(* CoDeSys 2.3.9.35 project: poka-yoke.pro *)
(* Author: Altus *)
(* Libraries: DU35x.lib 7.7.11 15:59:13, Navigation.lib 15.7.11 10:06:00, SysLibTargetVisu.lib 26.11.08 09:53:28, Standard.lib 26.11.08 09:46:20, Iecsfc.lib 26.11.08 09:46:14, SYSLIBCALLBACK.LIB 26.11.08 09:53:30 *)

(* PLC configuration (modules and I/O channels)
COM1 [COM1] node 0, in %IB0 out %QB0 {BaudRate = 115200; Paridade = Sem Paridade; StopBits = 1 Stop Bit; Modem = Sem RTS/CTS; Delay = 5}
  MToolIEC [Codesys] node 0, in %IB0 out %QB0
COM2 [COM2] node 1, in %IB0 out %QB0 {BaudRate = 115200; Paridade = Sem Paridade; StopBits = 1 Stop Bit; Modem = Sem RTS/CTS; Delay = 5}
  Desabilitada [Desabilitado485] node 0, in %IB0 out %QB0
Entradas Digitais 0 [Entradas0] node 0, in %IW0 out %QB0
  I00 AT %IX0.0 [BitInput] I0.0
  I01 AT %IX0.1 [BitInput] I0.1
  I02 AT %IX0.2 [BitInput] I0.2
  I03 AT %IX0.3 [BitInput] I0.3
  I04 AT %IX0.4 [BitInput] I0.4
  I05 AT %IX0.5 [BitInput] I0.5
  I06 AT %IX0.6 [BitInput] I0.6
  I07 AT %IX0.7 [BitInput] I0.7
  I08 AT %IX0.8 [BitInput] I0.8
Entradas Digitais 1 [Entradas1] node 0, in %IW1 out %QB0
  I10 AT %IX1.0 [BitInput] I1.0
  I11 AT %IX1.1 [BitInput] I1.1
  I12 AT %IX1.2 [BitInput] I1.2
  I13 AT %IX1.3 [BitInput] I1.3
  I14 AT %IX1.4 [BitInput] I1.4
  I15 AT %IX1.5 [BitInput] I1.5
  I16 AT %IX1.6 [BitInput] I1.6
  I17 AT %IX1.7 [BitInput] I1.7
  I18 AT %IX1.8 [BitInput] I1.8
I20 AT %IX2.0 [BitInput] I2.0
I21 AT %IX2.1 [BitInput] I2.1
AI0 AT %IW4 [WordInput] AI0 {TipoAnalogica = Channel Disable; FiltroAnalogica = Filter 0 - AI=2ms  / AV=90ms; FundoEscala = 0}
AI1 AT %IW5 [WordInput] AI1 {TipoAnalogica = Channel Disable; FiltroAnalogica = Filter 0 - AI=2ms  / AV=90ms; FundoEscala = 0}
AI2 AT %IW6 [WordInput] AI2 {TipoAnalogica = Channel Disable; FiltroAnalogica = Filter 0 - AI=2ms  / AV=90ms; FundoEscala = 0}
AI3 AT %IW7 [WordInput] AI3 {TipoAnalogica = Channel Disable; FiltroAnalogica = Filter 0 - AI=2ms  / AV=90ms; FundoEscala = 0}
Entradas Rápidas [EntradasRapidas] node 1, in %IB16 out %QB0
  Bloco 0 [Bloco0] node 0, in %IB16 out %QB0
    Desabilitado [DesabilitadoBloco0] node 0, in %IB16 out %QB0
  Bloco 1 [Bloco1] node 1, in %IB16 out %QB0
    Desabilitado [DesabilitadoBloco1] node 0, in %IB16 out %QB0
  Entrada Configuravél Bloco 0 [EntradaConfiBloco0] node 2, in %IB16 out %QB0
    Contador 0 [EntradaConfContador0] node 0, in %IB16 out %QB0 {EntradaConfiguravelContador = Disable}
  Entrada Configuravél Bloco 1 [EntradaConfiBloco1] node 3, in %IB16 out %QB0
    Contador 2 [EntradaConfContador2] node 0, in %IB16 out %QB0 {EntradaConfiguravelContador = Disable}
Saídas [Saidas] node 1, in %IB13 out %QB0
  Saídas Digitais 0 [Saidas0] node 0, in %IW0 out %QW0
    Q00 AT %QX0.0 [BitOutput] Q0.0
    Q01 AT %QX0.1 [BitOutput] Q0.1
    Q02 AT %QX0.2 [BitOutput] Q0.2
    Q03 AT %QX0.3 [BitOutput] Q0.3
    Q04 AT %QX0.4 [BitOutput] Q0.4
    Q05 AT %QX0.5 [BitOutput] Q0.5
    Q06 AT %QX0.6 [BitOutput] Q0.6
    Q07 AT %QX0.7 [BitOutput] Q0.7
  Saídas Digitais 1 [Saidas1] node 0, in %IW0 out %QW1
    Q10 AT %QX1.0 [BitOutput] Q1.0
    Q11 AT %QX1.1 [BitOutput] Q1.1
    Q12 AT %QX1.2 [BitOutput] Q1.2
    Q13 AT %QX1.3 [BitOutput] Q1.3
    Q14 AT %QX1.4 [BitOutput] Q1.4
    Q15 AT %QX1.5 [BitOutput] Q1.5
    Q16 AT %QX1.6 [BitOutput] Q1.6
    Q17 AT %QX1.7 [BitOutput] Q1.7
  Saídas Analógicas [SaidaAnalogica] node 0, in %IW0 out %QW3
    AO0 AT %QW3 [WordOutput] AO0 {TipoAnalogica = Channel Disable; FundoEscala = 0}
    AO1 AT %QW4 [WordOutput] AO1 {TipoAnalogica = Channel Disable; FundoEscala = 0}
  Saídas Rápidas [SaidasRapidas] node 1, in %IB0 out %QB10
    Saída Rápida 0 Desabilitada [DesabilitadoF0] node 0, in %IB0 out %QB10
    Saída Rápida 1 Desabilitada [DesabilitadoF1] node 1, in %IB0 out %QB10
  Saídas Comum de Contador [SaidasContador] node 2, in %IB0 out %QB10
    Saída do Bloco 0 Desabilitada [DesabilitadoSaidaBloco0] node 0, in %IB0 out %QB10
    Saída do Bloco 1 Desabilitada [DesabilitadoSaidaBloco1] node 1, in %IB0 out %QB10
Eventos Externos [Eventos] node 2, in %IB13 out %QB6
  Evento Temporizado [TimerEvent] node 0, in %IB13 out %QB6 {Intervalo = 10}
*)

(* Task configuration *)
TASK PRINCIPAL (PRIORITY := 1, INTERVAL := T#1ms);
	PLC_PRG();
END_TASK
TASK NAVIGATION (PRIORITY := 1, INTERVAL := T#20ms);
	NAVEGA();
END_TASK
TASK VISUALIZATION (PRIORITY := 1, INTERVAL := T#500ms);
	MAINTARGETVISU_PAINT_CODE
END_TASK
TASK KEYBOARD_USAGE (PRIORITY := 1, INTERVAL := T#20ms);
	MAINTARGETVISU_INPUT_CODE
END_TASK

(* Global variable list: Variáveis globais *)
(*CONSTANTES*)
VAR_GLOBAL CONSTANT
	NUMMAX_SENSORES: USINT := 14; (* NUMERO MAXIMO DE SENSORES *)
	NUMMAX_PARAFUSA: USINT := 1;
	NUMMAX_PROGBITS: USINT := 4;
	NUMMAX_MODELOS: USINT := 15;
	NUMMAX_SAIDAS: USINT := 14;
	NUM_ETAPAS: USINT := 12;
	NUM_ATIVOS: USINT := 4;
	SEGURANCA_ENABLED: BOOL := TRUE;
	CODE_PARAFUSA: USINT := 15;
	CODE_KEY_F: ARRAY [1..7] OF USINT := 16#70, 16#71, 16#72, 16#73, 16#74, 16#75, 16#76;
	CODE_KEY_MAIN: USINT := 16#24;
	CODE_KEY_UP: USINT := 16#26;
	CODE_KEY_DOWN: USINT := 16#28;
	CODE_KEY_DOT: USINT := 16#2E;
	CODE_KEY_ZERO: USINT := 16#30;
	CODE_KEY_ESC: USINT := 16#1B;
END_VAR

(*VARS GERAIS*)
VAR_GLOBAL
	PRIMEIRO_STEP: BOOL := TRUE;
	SEGUNDO_STEP: BOOL;
	TERCEIRO_STEP: BOOL;
	QUARTO_STEP: BOOL;
	QUINTO_STEP: BOOL;
	SEXTO_STEP: BOOL;
	SETIMO_STEP: BOOL;
	OITAVO_STEP: BOOL;
	NONO_STEP: BOOL;
	DECIMO_STEP: BOOL;
	ONZE_STEP: BOOL;
	DOZE_STEP: BOOL;
	TREZE_STEP: BOOL;
	QUATORZE_STEP: BOOL;
	QUINZE_STEP: BOOL;
	MODELOS_CONFIG4: BOOL;
	MODELOS_RANGE: USINT := 0;
	X: USINT := 1;
	Y: USINT := 1;
	Z: USINT := 1;
	IHM_X: USINT := 1;
	IHM_STRING_TITLE: STRING(20);
	IHM_STRING_DESCRIPTION: STRING(30);
	IHM_NUMMAX_SENSORES: USINT;
	IHM_NUMMAX_PARAFUSA: USINT;
	IHM_NUMMAX_PROGBITS: USINT;
	IHM_NUMMAX_PROGS: USINT;
	IHM_BLOQUEIA_PROGBITS: BOOL;
	IHM_BLOQUEIA_MODELOS: ARRAY [1..4] OF BOOL;
	IHM_ESCONDER_ZERAR: BOOL;
	IHM_ESCONDER_RESET: BOOL;
	IHM_ESCONDER_SETUP: BOOL;
	IHM_ESCONDER_MODELOS: ARRAY [1..4] OF BOOL;
	IHM_ESCONDER_MODELO4BACK: BOOL;
	IHM_ENTRADA_PROGS: BOOL;
	IHM_INT_ETAPAS: USINT;
	IHM_INT_ATIVOS: ARRAY [1..4] OF USINT;
	TECLA_F: ARRAY [1..7] OF BOOL;
	TECLA_MAIN: BOOL;
	TECLA_UP: BOOL;
	TECLA_DOWN: BOOL;
	TECLA_DOT: BOOL;
	TECLA_ZERO: BOOL;
	TECLA_ESC: BOOL;
	PASS_LIBERADO: BOOL;
	IHM_STRING_CHAVE: STRING(3);
	IHM_INT_SENHA: USINT;
	SENHA_GERADA : USINT;
	IHM_STRING_MODELOS: ARRAY [1..4] OF INT;
	MODELO_SELECIONADO: INT;

	(*MIGRADOS*)
	PRONTO: USINT;
	ARRAY_SENSORES_IN: ARRAY [1..NUMMAX_SENSORES] OF BOOL;
	ARRAY_SENSORES_OUT: ARRAY [1..NUMMAX_SENSORES] OF BOOL;
	ARRAY_SENSORES_OLDSTATE: ARRAY [1..NUMMAX_SENSORES] OF BOOL;
	ARRAY_DE_ATIVOS: ARRAY [1..NUM_ATIVOS] OF USINT;
	ARRAY_PROGBYTE_PARAFUSA: ARRAY [1..4] OF BOOL;
END_VAR

(*RETENTIVAS*)
VAR_GLOBAL RETAIN
	PRIMEIRO_START: BOOL := TRUE;
	NUM_SENSORES: USINT;
	NUM_PARAFUSA: USINT;
	NUM_PROGBITS: USINT;
	NUM_MODELOS: USINT;
	MATRIZ: ARRAY [1..NUMMAX_MODELOS, 1..NUM_ETAPAS, 1..NUM_ATIVOS] OF USINT;
	MODELOS: ARRAY [1..NUMMAX_MODELOS] OF INT;
END_VAR

(*VARS DE ENTRADA*)
VAR_GLOBAL (*--------VARIAVEIS DE ENTRADA-------*)
	KAP_IN 		AT %IX0.0: BOOL;
	SENSOR1_IN 	AT %IX0.1: BOOL;
	SENSOR2_IN 	AT %IX0.2: BOOL;
	SENSOR3_IN 	AT %IX0.3: BOOL;
	SENSOR4_IN 	AT %IX0.4: BOOL;
	SENSOR5_IN 	AT %IX0.5: BOOL;
	SENSOR6_IN 	AT %IX0.6: BOOL;
	SENSOR7_IN 	AT %IX0.7: BOOL;
	SENSOR8_IN 	AT %IX1.0: BOOL;
	SENSOR9_IN 	AT %IX1.1: BOOL;
	SENSOR10_IN AT %IX1.2: BOOL;
	TORQUEOK_IN AT %IX2.0: BOOL;
	TORQUENOK_IN AT %IX2.1: BOOL;
END_VAR

(*VARS DE SAIDA*)
VAR_GLOBAL
	SENSOR1_OUT AT %QX0.1: BOOL;
	SENSOR2_OUT AT %QX0.2: BOOL;
	SENSOR3_OUT AT %QX0.3: BOOL;
	SENSOR4_OUT AT %QX0.4: BOOL;
	SENSOR5_OUT AT %QX0.5: BOOL;
	SENSOR6_OUT AT %QX0.6: BOOL;
	SENSOR7_OUT AT %QX0.7: BOOL;
	SENSOR8_OUT AT %QX1.0: BOOL;
	SENSOR9_OUT AT %QX1.1: BOOL;
	SENSOR10_OUT AT %QX1.2: BOOL;
	PARAFUSA_ENABLE_OUT AT %QX1.3: BOOL;
	PARAFUSA_PROG1_OUT AT %QX1.4: BOOL;
	PARAFUSA_PROG2_OUT AT %QX1.5: BOOL;
	PARAFUSA_PROG3_OUT AT %QX1.6: BOOL;
	PARAFUSA_RESET_OUT AT %QX1.7: BOOL;
END_VAR

(* POU PLC_PRG, ST *)
PROGRAM PLC_PRG
VAR
	J: USINT; (* VAR USADA PARA LOOPS *)
	K: USINT; (* VAR USADA PARA LOOPS *)
	COUNT: USINT; (* VAR USADA PARA CONTAGENS *)
	NUMERO_ALEATORIO: USINT := 1;
	LETRA_ALEATORIA: STRING(1);
	NUMERO_2 : USINT := 10;
END_VAR

(*--INSTRUCOES DE MODIFICACAO
	EXPLICACOES DA PROGRAMACAO 
	COMENTARIOS ------------->*)
(*PRIMEIRA INICIALIZACAO - alternado*)
IF PRIMEIRO_STEP = TRUE  THEN
	IF PRIMEIRO_START = TRUE THEN
		IF J < 2 THEN (*RODA DUAS VEZES A INICIALIZACAO PARA GARANTIR*)
			PRG_INICIALIZA_VARS();
			CHANGE_SCREEN(ENABLE:=TRUE, VISU_NAME:='FIRST');
			J:= J +1;
		END_IF
		IF FUN_SCREEN_FIRST() = TRUE THEN
			PRIMEIRO_START := FALSE;
			CHANGE_SCREEN(ENABLE:=TRUE, VISU_NAME:='MAIN');
		END_IF
	ELSE
		PRIMEIRO_STEP := FALSE;
		SEGUNDO_STEP := TRUE;
		OITAVO_STEP := TRUE; (*talvez*)
		TECLA_F[4] := TRUE;
	END_IF
END_IF

(*CONFIGURA TELA MAIN - alternado*)
IF SEGUNDO_STEP = TRUE THEN
	(*ESCONDE BOTOES DE CONTROLE
	IHM_ESCONDER_ZERAR:= TRUE;
	IHM_ESCONDER_RESET:= TRUE;*)
	(*DEFINE OS MODELOS NA IHM*)
	FOR J:=1 TO 4 BY 1 DO
		IF J+MODELOS_RANGE <= NUM_MODELOS THEN
			IHM_STRING_MODELOS[J]:=MODELOS[J+MODELOS_RANGE];
		ELSE
			IHM_STRING_MODELOS[J]:=0;
		END_IF
	END_FOR
	(*ESCONDE OU MOSTRA O MODELO[4] NA IHM*)
	IF NUM_MODELOS = 4 THEN
		IHM_ESCONDER_MODELOS[4]:=FALSE;
		IHM_ESCONDER_MODELO4BACK:=FALSE;
		MODELOS_CONFIG4:=TRUE;
	ELSIF NUM_MODELOS > 4 THEN
		IHM_ESCONDER_MODELOS[4]:=TRUE;
		IHM_ESCONDER_MODELO4BACK:=TRUE;
		MODELOS_CONFIG4:=FALSE;
	ELSE
		IHM_ESCONDER_MODELOS[4]:=FALSE;
		IHM_ESCONDER_MODELO4BACK:=FALSE;
		MODELOS_CONFIG4:=FALSE;
	END_IF
	(*BLOQUEIA ENTRADA MODELOS IHM*)
	FOR J:=1 TO 4 BY 1 DO
		IHM_BLOQUEIA_MODELOS[J] := TRUE;
	END_FOR
	(*AVANÇA*)
	SEGUNDO_STEP:=FALSE;
	TERCEIRO_STEP:=TRUE;
	CHANGE_SCREEN(ENABLE:=TRUE, VISU_NAME:='PASS'); (*PARA DESBUGAR*)
	CHANGE_SCREEN(ENABLE:=TRUE, VISU_NAME:='MAIN'); (*ERRO DO CLP*)
	(*temp*)
	OITAVO_STEP := TRUE;
END_IF

(*VERIFICA KAP - continuo*)
IF TERCEIRO_STEP = TRUE THEN
	IF KAP_IN = TRUE THEN	(*= FALSE*)
		(*pausa tudo*)
		QUINZE_STEP := TRUE;
		IHM_STRING_TITLE := 'CONECTE';
		IHM_STRING_DESCRIPTION := 'KAP';
		IHM_ESCONDER_ZERAR:=TRUE;
		IHM_ESCONDER_RESET:=TRUE;
		IHM_ESCONDER_SETUP:=TRUE;
		QUINTO_STEP:=FALSE;
		SEXTO_STEP:=FALSE;
		NONO_STEP :=FALSE;
		DECIMO_STEP := FALSE;
	ELSE
		QUINTO_STEP := TRUE;
		SEXTO_STEP:=TRUE;
	END_IF
END_IF

(*ESCOLHA DO MODELO - continuo*)
IF QUINTO_STEP = TRUE THEN
	(*MOSTRA MAIS MODELOS*)
	IF IHM_ESCONDER_MODELO4BACK = TRUE THEN
		IF IsKeyPressed(CODE_KEY_F[7],0,0) = TRUE OR TECLA_F[7] = TRUE(*temp*) THEN
			IF MODELOS_RANGE < NUM_MODELOS -3 THEN
				MODELOS_RANGE := MODELOS_RANGE + 3;
			ELSE
				MODELOS_RANGE := 0;
			END_IF
			SEGUNDO_STEP:=TRUE;
		END_IF
	END_IF
	(*SELECIONA O MODELO*)
	FOR J:=1 TO 4 BY 1 DO
		IF IsKeyPressed(CODE_KEY_F[J+3],0,0) = TRUE OR TECLA_F[J+3] = TRUE(*temp*) THEN
			IF IHM_ESCONDER_MODELOS[J] = FALSE AND IHM_STRING_MODELOS[J] <> 0 THEN
				MODELO_SELECIONADO := IHM_STRING_MODELOS[J];
				IHM_ESCONDER_MODELOS[IHM_X] := FALSE;
				IHM_ESCONDER_MODELOS[J] := TRUE;
				IHM_X := J;
				X:= IHM_X + MODELOS_RANGE;
				Y:= 1;
				OITAVO_STEP := TRUE;
				PRG_SENSORES.DESATIVAR_TODOS();
				PRG_PARAFUSA.DESATIVAR();
				EXIT;
			END_IF
		END_IF
	END_FOR

	(*DESTACA MODELO SELECIONADO NA IHM*)
	IF MODELO_SELECIONADO <> IHM_STRING_MODELOS[IHM_X] THEN
		IHM_ESCONDER_MODELOS[IHM_X] := FALSE;
	ELSE
		IHM_ESCONDER_MODELOS[IHM_X] := TRUE;
	END_IF
	(*RESETA TECLAS - temp*)
	FOR J:=4 TO 7 BY 1 DO
		TECLA_F[J] := FALSE;(*temp*)
	END_FOR
END_IF

(*VERIFICA TECLAS DE CONTROLE - continuo*)
IF SEXTO_STEP = TRUE THEN
	IF IsKeyPressed(CODE_KEY_F[1],0,0) = TRUE OR TECLA_F[1] = TRUE(*temp*) THEN
		IF IHM_ESCONDER_ZERAR = FALSE THEN
			(*zera o ciclo*)
			PRG_SENSORES.DESATIVAR_TODOS();
			PRG_PARAFUSA.DESATIVAR();
			Y:= 1;
			OITAVO_STEP := TRUE;
		END_IF
		TECLA_F[1] := FALSE;(*temp*)
	END_IF
	IF IsKeyPressed(CODE_KEY_F[2],0,0) = TRUE OR TECLA_F[2] = TRUE(*temp*) THEN
		IF IHM_ESCONDER_RESET = FALSE THEN
			(*reseta do pause na etapa*)
			TERCEIRO_STEP := TRUE;
			QUINTO_STEP := TRUE;
			SEXTO_STEP := TRUE;
			DECIMO_STEP := TRUE;
		END_IF
		TECLA_F[2] := FALSE;(*temp*)
	END_IF
	IF IsKeyPressed(CODE_KEY_F[3],0,0) = TRUE OR TECLA_F[3] = TRUE(*temp*) THEN
		IF IHM_ESCONDER_SETUP = FALSE THEN
			(*desliga tudo e zera*)
			TERCEIRO_STEP := FALSE;
			QUINTO_STEP := FALSE;
			SEXTO_STEP := FALSE;
			(*vai para a tela PASS*)
			IF NUMERO_2 = 10 THEN
				LETRA_ALEATORIA := 'A';
			ELSIF NUMERO_2 = 11 THEN
				LETRA_ALEATORIA := 'B';
			ELSIF NUMERO_2 = 12 THEN
				LETRA_ALEATORIA := 'C';
			ELSIF NUMERO_2 = 13 THEN
				LETRA_ALEATORIA := 'D';
			ELSIF NUMERO_2 = 14 THEN
				LETRA_ALEATORIA := 'E';
			ELSIF NUMERO_2 = 15 THEN
				LETRA_ALEATORIA := 'F';
			END_IF
			IHM_STRING_CHAVE:= CONCAT(USINT_TO_STRING(NUMERO_ALEATORIO),LETRA_ALEATORIA);
			IHM_INT_SENHA := 0;
			SENHA_GERADA := NUMERO_ALEATORIO * NUMERO_2;
			CHANGE_SCREEN(ENABLE:=TRUE, VISU_NAME:='PASS');
			TREZE_STEP := TRUE;
		END_IF
		TECLA_F[3] := FALSE;(*temp*)
	END_IF
	IF IsKeyPressed(CODE_KEY_ZERO,0,0) = TRUE OR TECLA_ZERO = TRUE(*temp*) THEN
		(*desliga tudo e zera*)
		QUINZE_STEP := TRUE;
		NONO_STEP := FALSE;
		DECIMO_STEP := FALSE;
		TERCEIRO_STEP := FALSE;
		QUINTO_STEP := FALSE;
		SEXTO_STEP := FALSE;
		QUATORZE_STEP := TRUE;
		IHM_ESCONDER_MODELOS[IHM_X] := FALSE;
		(*habilita entrada edit modelos*)
		IHM_STRING_TITLE := 'MODO';
		IHM_STRING_DESCRIPTION := 'EDIÇÃO';
		FOR J:=1 TO 4 BY 1 DO
			IF IHM_STRING_MODELOS[J] <> 0 THEN
				IHM_BLOQUEIA_MODELOS[J] := FALSE;
			END_IF
		END_FOR
		IF IHM_ESCONDER_MODELO4BACK = TRUE THEN
			IHM_BLOQUEIA_MODELOS[4] := TRUE;
		END_IF
		CHANGE_SCREEN(ENABLE:=TRUE, VISU_NAME:='PASS'); (*PARA DESBUGAR*)
		CHANGE_SCREEN(ENABLE:=TRUE, VISU_NAME:='MAIN'); (*ERRO DO CLP*)
		TECLA_ZERO := FALSE;
	END_IF
END_IF

(*CONTROLE DA TELA SETUP - alternado*)
IF SETIMO_STEP = TRUE THEN
	IF FUN_SCREEN_SETUP() = TRUE THEN
		CHANGE_SCREEN(ENABLE:=TRUE, VISU_NAME:='MAIN');
		SETIMO_STEP:=FALSE;
		TERCEIRO_STEP := TRUE;
		QUINTO_STEP := TRUE;
		SEXTO_STEP := TRUE;
		OITAVO_STEP:= TRUE;
		(*ativa steps*)
	END_IF
	IF IsKeyPressed(CODE_KEY_DOT,0,0) = TRUE OR TECLA_DOT = TRUE(*temp*) THEN
		(*vai para a tela FIRST*)
		CHANGE_SCREEN(ENABLE:=TRUE, VISU_NAME:='FIRST');
		SETIMO_STEP := FALSE;
		DOZE_STEP := TRUE;
		TECLA_DOT:= FALSE;
	END_IF
END_IF

(*VERIFICA MATRIZ ANTES DE INICIAR CICLO - alternado*)
IF OITAVO_STEP = TRUE THEN
	COUNT:=0;
	FOR J:=1 TO NUM_ETAPAS BY 1 DO
		FOR K:=1 TO NUM_ATIVOS -1 BY 1 DO
			IF MATRIZ[X,J,K] = 0 THEN
				COUNT:= COUNT +1;
			END_IF
		END_FOR
	END_FOR
	IF COUNT = (NUM_ETAPAS * (NUM_ATIVOS -1)) THEN
		IHM_ESCONDER_ZERAR := TRUE;
		IHM_ESCONDER_RESET := TRUE;
		DECIMO_STEP := FALSE;
		NONO_STEP := FALSE;
		IHM_STRING_TITLE:= 'CADASTRAR';
		IHM_STRING_DESCRIPTION:= 'MODELO';
	ELSE
		IHM_ESCONDER_ZERAR := FALSE;
		IHM_ESCONDER_RESET := FALSE;
		IHM_STRING_TITLE:= '';	(*talvez*)
		IHM_STRING_DESCRIPTION:= 'OK';	(*talvez*)
		NONO_STEP:=TRUE;
	END_IF
	OITAVO_STEP := FALSE;
END_IF

(*ATIVA DEVICES*)
IF NONO_STEP = TRUE THEN
	(*FOR Z:=1 TO NUM_ATIVOS -1 BY 1 DO  ---- NOVO
		IF MATRIZ[X,Y,Z] <> 0 THEN
			IF MATRIZ[X,Y,Z] = CODE_PARAFUSA THEN
				PRG_PARAFUSA.ATIVAR();
			ELSE
				PRG_SENSORES.ATIVAR();
			END_IF
		END_IF
	END_FOR
	PRG_UPDATE_OUT;*)
	IF Y > NUM_ETAPAS THEN
		Y := 1;
	END_IF
	FOR Z:=1 TO NUM_ATIVOS BY 1 DO
		ARRAY_DE_ATIVOS[Z] := MATRIZ[X,Y,Z];
	END_FOR
	FOR Z:=1 TO NUM_ATIVOS-1 BY 1 DO
		IF ARRAY_DE_ATIVOS[Z] <> 0 THEN
			IF ARRAY_DE_ATIVOS[Z] = CODE_PARAFUSA THEN
				(*PARAFUSA_PROG := ARRAY_DE_ATIVOS[NUM_ATIVOS];*)
				PRG_PARAFUSA.ATIVAR();
			ELSE
				(*SENSOR_ALVO := ARRAY_DE_ATIVOS[Z];*)
				PRG_SENSORES.ATIVAR();
			END_IF
		END_IF
	END_FOR
	NONO_STEP := FALSE;
	DECIMO_STEP := TRUE;
END_IF

(*LOOP DE VERIFICAÇÃO DOS DEVICES*)
IF DECIMO_STEP = TRUE THEN
	PRONTO := 0;
	IHM_STRING_TITLE := 'ATIVOS';
	IHM_STRING_DESCRIPTION := '';
	FOR Z:=1 TO NUM_ATIVOS -1 BY 1 DO
		IF ARRAY_DE_ATIVOS[Z] <> 0 THEN
			IF ARRAY_DE_ATIVOS[Z] = CODE_PARAFUSA THEN
				IHM_STRING_DESCRIPTION := CONCAT(IHM_STRING_DESCRIPTION, ' P');
				IHM_STRING_DESCRIPTION := CONCAT(IHM_STRING_DESCRIPTION, USINT_TO_STRING(ARRAY_DE_ATIVOS[4]));
				PRG_PARAFUSA.TORQUE();
				IF PRG_PARAFUSA.ERRO = TRUE THEN
					IHM_STRING_TITLE := 'PEÇA';
					IHM_STRING_DESCRIPTION := 'ERRADA';
					QUINZE_STEP := TRUE;
					EXIT;
				END_IF
			ELSE
				IHM_STRING_DESCRIPTION := CONCAT(IHM_STRING_DESCRIPTION, ' S');
				IHM_STRING_DESCRIPTION := CONCAT(IHM_STRING_DESCRIPTION, USINT_TO_STRING(ARRAY_DE_ATIVOS[Z]));
				PRG_SENSORES.READTODOS();
				IF PRG_SENSORES.ERRO = TRUE THEN
					IHM_STRING_TITLE := 'PEÇA';
					IHM_STRING_DESCRIPTION := 'ERRADA';
					QUINZE_STEP := TRUE;
					EXIT;
				END_IF
			END_IF
		ELSE
			PRONTO := PRONTO + 1;
		END_IF
	END_FOR
	IF PRONTO = 3 THEN
		Y := Y+1;
		DECIMO_STEP := FALSE;
		NONO_STEP := TRUE;
	END_IF
END_IF

(*RESETA TECLAS PARA EVITAR ERRO EM TELAS SETUP E FIRST*)
(*IF ONZE_STEP = TRUE THEN*)
IF QUINTO_STEP = FALSE OR SEXTO_STEP = FALSE THEN (*validar aplicação*)
	IsKeyPressed(CODE_KEY_F[1],0,0);
	IsKeyPressed(CODE_KEY_F[2],0,0);
	IsKeyPressed(CODE_KEY_F[3],0,0);
	IsKeyPressed(CODE_KEY_F[4],0,0);
	IsKeyPressed(CODE_KEY_F[5],0,0);
	IsKeyPressed(CODE_KEY_F[6],0,0);
	IsKeyPressed(CODE_KEY_F[7],0,0);
	IsKeyPressed(CODE_KEY_DOT,0,0);
END_IF

(*CONTROLE DA TELA FIRST - alternado*)
IF DOZE_STEP = TRUE THEN
	IF FUN_SCREEN_FIRST() = TRUE THEN
		CHANGE_SCREEN(ENABLE:=TRUE, VISU_NAME:='MAIN');
		DOZE_STEP:=FALSE;
		SEGUNDO_STEP:= TRUE;
		QUINTO_STEP := TRUE;
		SEXTO_STEP := TRUE;
		OITAVO_STEP:= TRUE;
		NONO_STEP := TRUE;
		(*volta para modelo 1*)
		MODELOS_RANGE:= 0;
		TECLA_F[4] := TRUE;
	END_IF
END_IF

(*CONTROLE DA TELA PASS - alternado*)
IF TREZE_STEP = TRUE THEN
	IF SEGURANCA_ENABLED = TRUE THEN
		IF FUN_SCREEN_PASS() = TRUE THEN
			IF PASS_LIBERADO = TRUE THEN
				QUINZE_STEP := TRUE;
				NONO_STEP:= FALSE;
				DECIMO_STEP := FALSE;
				(*inicializa vars da tela setup*)
				IHM_INT_ETAPAS := 1;
				FOR J:=1 TO 4 BY 1 DO
				IHM_INT_ATIVOS[J] := MATRIZ[X, IHM_INT_ETAPAS, J];
				END_FOR
				CHANGE_SCREEN(ENABLE:=TRUE, VISU_NAME:='SETUP');
				SETIMO_STEP := TRUE;
			ELSE
				(*volta para o main*)
				CHANGE_SCREEN(ENABLE:=TRUE, VISU_NAME:='MAIN');
				TERCEIRO_STEP := TRUE;
				QUINTO_STEP := TRUE;
				SEXTO_STEP := TRUE;
				OITAVO_STEP:= TRUE;
			END_IF
			TREZE_STEP := FALSE;
		END_IF
	ELSE
		(*inicializa vars da tela setup*)
		IHM_INT_ETAPAS := 1;
		FOR J:=1 TO 4 BY 1 DO
			IHM_INT_ATIVOS[J] := MATRIZ[X, IHM_INT_ETAPAS, J];
		END_FOR
		CHANGE_SCREEN(ENABLE:=TRUE, VISU_NAME:='SETUP');
		SETIMO_STEP := TRUE;
		TREZE_STEP := FALSE;
	END_IF
END_IF

(*CONTROLE EDICAO NOME DOS MODELOS*)
IF QUATORZE_STEP = TRUE THEN
	IF FUN_EDITA_MODELOS() = TRUE THEN
		MODELO_SELECIONADO := MODELOS[X];
		(*volta para o main*)
		CHANGE_SCREEN(ENABLE:=TRUE, VISU_NAME:='MAIN');
		SEGUNDO_STEP := TRUE;
		TERCEIRO_STEP := TRUE;
		QUINTO_STEP := TRUE;
		SEXTO_STEP := TRUE;
		OITAVO_STEP:= TRUE;
		QUATORZE_STEP := FALSE;
	END_IF
END_IF

(*CASO DE EM RESET*)
IF QUINZE_STEP = TRUE THEN
	PRG_SENSORES.DESATIVAR_TODOS();
	PRG_PARAFUSA.DESATIVAR();
	NONO_STEP:=FALSE;
	DECIMO_STEP:=FALSE;
	QUINZE_STEP := FALSE;
END_IF


(*GERADOR DO NUMERO ALEATORIO*)
IF NUMERO_ALEATORIO < 3 THEN
	NUMERO_ALEATORIO := NUMERO_ALEATORIO +1;
ELSE
	NUMERO_ALEATORIO := 1;
END_IF
(*GERADOR DO NUMERO_2*)
IF NUMERO_2 < 15 THEN
	NUMERO_2 := NUMERO_2 +1;
ELSE
	NUMERO_2 := 10;
END_IF
IF (NUMERO_ALEATORIO * (NUMERO_2 -10)) = 6 THEN
	NUMERO_2 := NUMERO_2 +1;
END_IF
END_PROGRAM

(* POU PRG_INICIALIZA_VARS, ST *)
PROGRAM PRG_INICIALIZA_VARS
VAR
	J: INT;
END_VAR
(*INIT PARA IHM FIRST*)
NUM_SENSORES:=10;
NUM_PARAFUSA:=1;
NUM_PROGBITS:=3;
NUM_MODELOS :=6;

(*INIT DA MATRIZ DAS SEQUENCIAS - temp*)
MATRIZ[1,1,1]:= 1;
MATRIZ[1,1,2]:= 3;
MATRIZ[1,1,3]:= 7;
MATRIZ[1,2,1]:= 4;
MATRIZ[1,2,2]:= 5;
MATRIZ[1,3,1]:= 6;
MATRIZ[1,3,2]:= 2;
MATRIZ[1,3,3]:= 15;
MATRIZ[1,3,4]:= 2;

(*INIT TODOS MODELOS*)
FOR J:=1 TO NUMMAX_MODELOS BY 1 DO
	MODELOS[J]:=1000+J;
END_FOR

(*INIT PARA IHM MAIN*)
MODELO_SELECIONADO := MODELOS[1];
IHM_ESCONDER_MODELOS[1] := TRUE;
END_PROGRAM

(* POU FUN_SCREEN_FIRST, ST *)
FUNCTION FUN_SCREEN_FIRST : BOOL
VAR_INPUT
END_VAR
VAR
END_VAR
(*VERIFICA A TECLA F7 PARA ENCERRAR A TELA FIRST*)
IF IsKeyPressed(CODE_KEY_F[7],0,0) = TRUE OR TECLA_F[7] = TRUE (*debug*) OR
IsKeyPressed(CODE_KEY_MAIN,0,0) = TRUE OR TECLA_MAIN = TRUE (*debug*) THEN
	TECLA_F[7] := FALSE; (*debug*)
	TECLA_MAIN := FALSE; (*debug*)
	FUN_SCREEN_FIRST:=TRUE;
	RETURN;
END_IF

(*CORRIGE OS BOTOES UP E DOWN PARA NAO SAIR DA TELA FIRST*)
IF IsKeyPressed(CODE_KEY_UP,0,0) = TRUE OR TECLA_UP = TRUE (*debug*) OR
IsKeyPressed(CODE_KEY_DOWN,0,0) = TRUE OR TECLA_DOWN = TRUE (*debug*) THEN
	TECLA_UP := FALSE; (*debug*)
	TECLA_DOWN := FALSE; (*debug*)
	CHANGE_SCREEN(ENABLE:=TRUE, VISU_NAME:='FIRST');
END_IF

(*DETERMINA O NUMERO MAXIMO DE SENSORES*)
IHM_NUMMAX_SENSORES := NUMMAX_SAIDAS - (NUM_PARAFUSA + NUM_PROGBITS);

(*DETERMINA O NUMERO MAXIMO DE PARAFUSADEIRA*)
IF NUM_SENSORES < NUMMAX_SAIDAS-1 THEN
	IHM_NUMMAX_PARAFUSA:= 1;
ELSE
	IHM_NUMMAX_PARAFUSA:= 0;
END_IF

(*DETERMINA O NUMERO MAXIMO DE PROGBITS*)
IF NUM_PARAFUSA = 0 THEN
	IHM_BLOQUEIA_PROGBITS := TRUE;
	NUM_PROGBITS := 0;
ELSE
	IHM_BLOQUEIA_PROGBITS := FALSE;
	IF NUM_PROGBITS = 0 THEN
		NUM_PROGBITS:= NUMMAX_SAIDAS-1 -NUM_SENSORES;
		IF NUM_PROGBITS > NUMMAX_PROGBITS THEN
			NUM_PROGBITS := NUMMAX_PROGBITS;
		END_IF
	END_IF
	IHM_NUMMAX_PROGBITS := NUMMAX_SAIDAS-1 -NUM_SENSORES;
	IF IHM_NUMMAX_PROGBITS > NUMMAX_PROGBITS THEN
		IHM_NUMMAX_PROGBITS := NUMMAX_PROGBITS;
	END_IF
END_IF
END_FUNCTION

(* POU PRG_SENSORES, ST *)
PROGRAM PRG_SENSORES
VAR
	ERRO: BOOL;
	J: USINT;
	K: USINT;
	ACHOU: BOOL;
END_VAR
RETURN;
END_PROGRAM
ACTION ATIVAR:
IF ARRAY_DE_ATIVOS[Z] <> 0 THEN
	ARRAY_SENSORES_OUT[ARRAY_DE_ATIVOS[Z]] := TRUE;
END_IF
UPDATE_OUT();
RETURN;
END_ACTION
ACTION DESATIVAR_TODOS:
FOR J:=1 TO NUM_SENSORES BY 1 DO
	ARRAY_SENSORES_OUT[J] := FALSE;
	ARRAY_SENSORES_OLDSTATE[J] := FALSE;
END_FOR
UPDATE_OUT();
RETURN;
END_ACTION
ACTION READTODOS:
UPDATE_IN();
ERRO := FALSE;
FOR J:=1 TO NUM_SENSORES BY 1 DO
	IF ARRAY_SENSORES_IN[J] = TRUE AND ARRAY_SENSORES_OLDSTATE[J] = FALSE THEN
		ACHOU := FALSE;
		FOR K:=1 TO NUM_ATIVOS-1 BY 1 DO
			IF ARRAY_DE_ATIVOS[K] <> 0 THEN
				IF J = ARRAY_DE_ATIVOS[K] THEN
					ARRAY_SENSORES_OLDSTATE[J] := TRUE;
					ACHOU := TRUE;
					EXIT;
				END_IF
			END_IF
		END_FOR
		IF ACHOU <> TRUE THEN
			ERRO := TRUE;
			EXIT;
		END_IF
	END_IF
	IF ARRAY_SENSORES_IN[J] = FALSE AND ARRAY_SENSORES_OLDSTATE[J] = TRUE THEN
		ARRAY_SENSORES_OUT[J] := FALSE;
		ARRAY_SENSORES_OLDSTATE[J] := FALSE;
		FOR K:=1 TO NUM_ATIVOS-1 BY 1 DO
			IF J = ARRAY_DE_ATIVOS[K] THEN
				ARRAY_DE_ATIVOS[K] := 0;
			END_IF
		END_FOR
	END_IF
END_FOR
UPDATE_OUT();
RETURN;
END_ACTION
ACTION UPDATE_IN:
ARRAY_SENSORES_IN[1] := SENSOR1_IN;
ARRAY_SENSORES_IN[2] := SENSOR2_IN;
ARRAY_SENSORES_IN[3] := SENSOR3_IN;
ARRAY_SENSORES_IN[4] := SENSOR4_IN;
ARRAY_SENSORES_IN[5] := SENSOR5_IN;
ARRAY_SENSORES_IN[6] := SENSOR6_IN;
ARRAY_SENSORES_IN[7] := SENSOR7_IN;
ARRAY_SENSORES_IN[8] := SENSOR8_IN;
ARRAY_SENSORES_IN[9] := SENSOR9_IN;
ARRAY_SENSORES_IN[10] := SENSOR10_IN;
RETURN;
END_ACTION
ACTION UPDATE_OUT:
SENSOR1_OUT := ARRAY_SENSORES_OUT[1];
SENSOR2_OUT := ARRAY_SENSORES_OUT[2];
SENSOR3_OUT := ARRAY_SENSORES_OUT[3];
SENSOR4_OUT := ARRAY_SENSORES_OUT[4];
SENSOR5_OUT := ARRAY_SENSORES_OUT[5];
SENSOR6_OUT := ARRAY_SENSORES_OUT[6];
SENSOR7_OUT := ARRAY_SENSORES_OUT[7];
SENSOR8_OUT := ARRAY_SENSORES_OUT[8];
SENSOR9_OUT := ARRAY_SENSORES_OUT[9];
SENSOR10_OUT := ARRAY_SENSORES_OUT[10];
RETURN;
END_ACTION

(* POU PRG_PARAFUSA, ST *)
PROGRAM PRG_PARAFUSA
VAR
	ERRO: BOOL;
END_VAR
RETURN;
END_PROGRAM
ACTION ATIVAR:
CASE ARRAY_DE_ATIVOS[NUM_ATIVOS] OF
	1:	ARRAY_PROGBYTE_PARAFUSA[1] := FALSE;
		ARRAY_PROGBYTE_PARAFUSA[2] := FALSE;
		ARRAY_PROGBYTE_PARAFUSA[3] := TRUE;
	2:	ARRAY_PROGBYTE_PARAFUSA[1] := FALSE;
		ARRAY_PROGBYTE_PARAFUSA[2] := TRUE;
		ARRAY_PROGBYTE_PARAFUSA[3] := FALSE;
	3:	ARRAY_PROGBYTE_PARAFUSA[1] := FALSE;
		ARRAY_PROGBYTE_PARAFUSA[2] := TRUE;
		ARRAY_PROGBYTE_PARAFUSA[3] := TRUE;
	4:	ARRAY_PROGBYTE_PARAFUSA[1] := TRUE;
		ARRAY_PROGBYTE_PARAFUSA[2] := FALSE;
		ARRAY_PROGBYTE_PARAFUSA[3] := FALSE;
	5:	ARRAY_PROGBYTE_PARAFUSA[1] := TRUE;
		ARRAY_PROGBYTE_PARAFUSA[2] := FALSE;
		ARRAY_PROGBYTE_PARAFUSA[3] := TRUE;
	6:	ARRAY_PROGBYTE_PARAFUSA[1] := TRUE;
		ARRAY_PROGBYTE_PARAFUSA[2] := FALSE;
	7:	ARRAY_PROGBYTE_PARAFUSA[1] := TRUE;
		ARRAY_PROGBYTE_PARAFUSA[2] := TRUE;
		ARRAY_PROGBYTE_PARAFUSA[3] := TRUE;
END_CASE
PARAFUSA_RESET_OUT := FALSE;
PARAFUSA_PROG1_OUT := ARRAY_PROGBYTE_PARAFUSA[1];
PARAFUSA_PROG2_OUT := ARRAY_PROGBYTE_PARAFUSA[2];
PARAFUSA_PROG3_OUT := ARRAY_PROGBYTE_PARAFUSA[3];
PARAFUSA_ENABLE_OUT := TRUE;
RETURN;
END_ACTION
ACTION DESATIVAR:
PARAFUSA_RESET_OUT := FALSE;
PARAFUSA_ENABLE_OUT := FALSE;
PARAFUSA_PROG1_OUT := FALSE;
PARAFUSA_PROG2_OUT := FALSE;
PARAFUSA_PROG3_OUT := FALSE;
RETURN;
END_ACTION
ACTION TORQUE:
ERRO := FALSE;
IF TORQUEOK_IN = TRUE THEN
	ARRAY_DE_ATIVOS[Z] := 0;
	PARAFUSA_ENABLE_OUT := FALSE;
	PARAFUSA_PROG1_OUT := FALSE;
	PARAFUSA_PROG2_OUT := FALSE;
	PARAFUSA_PROG3_OUT := FALSE;
	ERRO:= FALSE;
END_IF
IF TORQUENOK_IN = TRUE THEN
	PARAFUSA_ENABLE_OUT := FALSE;
	PARAFUSA_RESET_OUT := TRUE;
	ERRO:= TRUE;
END_IF
RETURN;
END_ACTION

(* POU FUN_SCREEN_SETUP, ST *)
FUNCTION FUN_SCREEN_SETUP : BOOL
VAR_INPUT
END_VAR
VAR
	J: USINT;
	K: USINT;
	C: USINT;
	HAVE: BOOL;
END_VAR
(*VERIFICA A TECLA MAIN PARA ENCERRAR A TELA SETUP*)
IF IsKeyPressed(CODE_KEY_F[7],0,0) = TRUE OR TECLA_F[7] = TRUE (*debug*) OR
IsKeyPressed(CODE_KEY_MAIN,0,0) = TRUE OR TECLA_MAIN = TRUE (*debug*) THEN
	TECLA_F[7] := FALSE; (*debug*)
	TECLA_MAIN := FALSE; (*debug*)
	FUN_SCREEN_SETUP:=TRUE;
	RETURN;
END_IF

(*TECLA UP - DECREMENTA ETAPA MOSTRADA*)
IF IsKeyPressed(CODE_KEY_UP,0,0) = TRUE OR TECLA_UP = TRUE(*temp*) THEN
	IF IHM_INT_ETAPAS > 1 THEN
		IHM_INT_ETAPAS := IHM_INT_ETAPAS - 1;
		FOR J:=1 TO 4 BY 1 DO
			IHM_INT_ATIVOS[J] := MATRIZ[X, IHM_INT_ETAPAS, J];
		END_FOR
	END_IF
	TECLA_UP := FALSE; (*temp*)
	CHANGE_SCREEN(ENABLE:=TRUE, VISU_NAME:='FIRST'); (*PARA DESBUGAR*)
	CHANGE_SCREEN(ENABLE:=TRUE, VISU_NAME:='SETUP'); (*ERRO DO CLP*)
END_IF

(*TECLA DOWN - INCREMENTA ETAPA MOSTRADA*)
IF IsKeyPressed(CODE_KEY_DOWN,0,0) = TRUE OR TECLA_DOWN = TRUE(*temp*) THEN
	IF IHM_INT_ETAPAS < NUM_ETAPAS THEN
		IHM_INT_ETAPAS := IHM_INT_ETAPAS + 1;
		FOR J:=1 TO 4 BY 1 DO
			IHM_INT_ATIVOS[J] := MATRIZ[X, IHM_INT_ETAPAS, J];
		END_FOR
	END_IF
	TECLA_DOWN := FALSE; (*temp*)
	CHANGE_SCREEN(ENABLE:=TRUE, VISU_NAME:='FIRST'); (*PARA DESBUGAR*)
	CHANGE_SCREEN(ENABLE:=TRUE, VISU_NAME:='SETUP'); (*ERRO DO CLP*)
END_IF

(*VALIDA OS VALORES DOS ATIVOS*)
FOR J:=1 TO 3 BY 1 DO
	IF IHM_INT_ATIVOS[J] > NUM_SENSORES AND IHM_INT_ATIVOS[J] <> 15 THEN
		IHM_INT_ATIVOS[J] := NUM_SENSORES;
	END_IF
	IF IHM_INT_ATIVOS[J] = CODE_PARAFUSA THEN
		HAVE := TRUE;
		IF NUM_PARAFUSA = 0 THEN
			IHM_INT_ATIVOS[J] := 0;
		END_IF
	END_IF
	C:=0;
	FOR K:=1 TO 3 BY 1 DO
		IF IHM_INT_ATIVOS[J] = IHM_INT_ATIVOS[K] AND IHM_INT_ATIVOS[K] <> 0 THEN
			C := C +1;
			IF C > 1 THEN
				IHM_INT_ATIVOS[K]:= 0;
			END_IF
		END_IF
	END_FOR
END_FOR
IF HAVE = FALSE THEN
	IHM_INT_ATIVOS[4] := 0;
	IHM_ENTRADA_PROGS:= TRUE;
ELSE
	IHM_ENTRADA_PROGS:= FALSE;
END_IF
IF NUM_PROGBITS = 0 THEN
	IHM_ENTRADA_PROGS:= TRUE;
END_IF
IHM_NUMMAX_PROGS:= REAL_TO_USINT(EXPT(2,NUM_PROGBITS)) -1;
IF IHM_INT_ATIVOS[4] > IHM_NUMMAX_PROGS THEN
	IHM_INT_ATIVOS[4] := 0;
END_IF

(*ESCREVE OS VALORES DA TELA NA MATRIZ*)
FOR J:=1 TO 4 BY 1 DO
	MATRIZ[X, IHM_INT_ETAPAS, J] := IHM_INT_ATIVOS[J];
END_FOR
END_FUNCTION

(* POU FUN_SCREEN_PASS, ST *)
FUNCTION FUN_SCREEN_PASS : BOOL
VAR_INPUT
END_VAR
VAR
END_VAR
(*VERIFICA A TECLA F7 PARA ENCERRAR A TELA PASS*)
IF IsKeyPressed(CODE_KEY_F[7],0,0) = TRUE OR TECLA_F[7] = TRUE (*debug*) OR
IsKeyPressed(CODE_KEY_MAIN,0,0) = TRUE OR TECLA_MAIN = TRUE (*debug*) THEN
	TECLA_F[7] := FALSE; (*debug*)
	TECLA_MAIN := FALSE; (*debug*)
	PASS_LIBERADO := FALSE;
	FUN_SCREEN_PASS:=TRUE;
	RETURN;
END_IF

(*CORRIGE OS BOTOES UP E DOWN PARA NAO SAIR DA TELA PASS*)
IF IsKeyPressed(CODE_KEY_UP,0,0) = TRUE OR TECLA_UP = TRUE (*debug*) OR
IsKeyPressed(CODE_KEY_DOWN,0,0) = TRUE OR TECLA_DOWN = TRUE (*debug*) THEN
	TECLA_UP := FALSE; (*debug*)
	TECLA_DOWN := FALSE; (*debug*)
	CHANGE_SCREEN(ENABLE:=TRUE, VISU_NAME:='PASS');
END_IF

IF IHM_INT_SENHA <> 0 THEN
	IF IHM_INT_SENHA = SENHA_GERADA THEN
		PASS_LIBERADO := TRUE;
		FUN_SCREEN_PASS:=TRUE;
	ELSE
		PASS_LIBERADO := FALSE;
		FUN_SCREEN_PASS:=TRUE;
	END_IF
END_IF
END_FUNCTION

(* POU FUN_EDITA_MODELOS, ST *)
FUNCTION FUN_EDITA_MODELOS : BOOL
VAR_INPUT
END_VAR
VAR
	J: USINT; K: USINT; COUNT:USINT;
END_VAR
IF IsKeyPressed(CODE_KEY_ESC,0,0) = TRUE OR TECLA_ESC = TRUE (*debug*) OR
IsKeyPressed(CODE_KEY_MAIN,0,0) = TRUE OR TECLA_MAIN = TRUE (*debug*) THEN
	TECLA_ESC := FALSE; (*debug*)
	TECLA_MAIN := FALSE; (*debug*)
	FUN_EDITA_MODELOS:=TRUE;
	RETURN;
END_IF

FOR J:=1 TO 3 BY 1 DO
	IF IHM_STRING_MODELOS[J] <> 0 THEN
		MODELOS[J+MODELOS_RANGE] := IHM_STRING_MODELOS[J];
	END_IF
END_FOR

IF IHM_ESCONDER_MODELO4BACK = FALSE THEN
	IF IHM_STRING_MODELOS[4] <> 0 THEN
		MODELOS[4] := IHM_STRING_MODELOS[4];
	END_IF
END_IF

FOR J:=1 TO NUM_MODELOS BY 1 DO
	COUNT := 0;
	FOR K:=1 TO NUM_MODELOS BY 1 DO
		IF MODELOS[J] = MODELOS[K] THEN
			COUNT := COUNT +1;
			IF COUNT > 1 THEN
				MODELOS[K] := 9990+K;
				EXIT;
			END_IF
		END_IF
	END_FOR
END_FOR
END_FUNCTION

(* POU NAVEGA, ST *)
PROGRAM NAVEGA
VAR
	ControleTelas : NAVIGATION;
	ListaTelas 	: ARRAY [0..30] OF STRING(10);
END_VAR
(* Adiciona a tela MAIN como tela principal *)
ListaTelas[0] := 'MAIN';

(* Ativa o controle automático de navegação somente pelo teclado *)
ControleTelas(ENABLE_UPDW := FALSE, VISU_LIST := ListaTelas, UP := FALSE , DOWN := FALSE);
END_PROGRAM

(* POU DEF_MODELO, ST *)
PROGRAM DEF_MODELO
VAR
END_VAR
MODELO_SELECIONADO := IHM_STRING_MODELOS[IHM_X];
IHM_ESCONDER_MODELOS[IHM_X] := FALSE;
X:= IHM_X + MODELOS_RANGE;
Y:= 1;
OITAVO_STEP:= TRUE;
END_PROGRAM

(* POU PRG_UPDATE_IN, ST *)
PROGRAM PRG_UPDATE_IN
VAR
END_VAR
X:=X;
END_PROGRAM

(* POU PRG_UPDATE_OUT, ST *)
PROGRAM PRG_UPDATE_OUT
VAR
END_VAR
X:=X;
END_PROGRAM

(* Visualisation FIRST
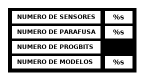
rectangle at (3,2)-(93,16): text "NUMERO DE SENSORES"
rectangle at (3,17)-(93,31): text "NUMERO DE PARAFUSA"
rectangle at (3,32)-(93,46): text "NUMERO DE PROGBITS"
rectangle at (96,2)-(125,16): text "%s"; shows .NUM_SENSORES; editable 1...IHM_NUMMAX_SENSORES
rectangle at (96,17)-(125,31): text "%s"; shows .NUM_PARAFUSA; editable 0...IHM_NUMMAX_PARAFUSA
rectangle at (3,47)-(93,61): text "NUMERO DE MODELOS"
rectangle at (96,47)-(125,61): text "%s"; shows .NUM_MODELOS; editable 1...NUMMAX_MODELOS
1 more shapes without text or variables
1 elements of other kinds (tables, trends, ...) not read
*)

(* Visualisation MAIN
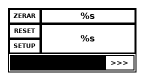
rectangle at (1,1)-(32,15): text "----"
rectangle at (1,16)-(32,30): text "----"
rectangle at (33,16)-(127,45): text "%s"; shows .IHM_STRING_DESCRIPTION
rectangle at (33,1)-(127,15): text "%s"; shows .IHM_STRING_TITLE
rectangle at (1,1)-(32,15): text "ZERAR"; invisible if .IHM_ESCONDER_ZERAR
rectangle at (1,16)-(32,30): text "RESET"; invisible if .IHM_ESCONDER_RESET
rectangle at (97,47)-(126,62): text ">>>"
rectangle at (1,31)-(32,45): text "----"
rectangle at (1,31)-(32,45): text "SETUP"; invisible if .IHM_ESCONDER_SETUP
2 more shapes without text or variables
8 elements of other kinds (tables, trends, ...) not read
*)

(* Visualisation PASS
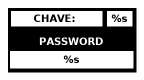
rectangle at (2,2)-(95,19): text "CHAVE:"
rectangle at (98,2)-(125,19): text "%s"; shows IHM_STRING_CHAVE
rectangle at (22,25)-(105,42): text "PASSWORD"
rectangle at (2,43)-(125,60): text "%s"; shows .IHM_INT_SENHA; editable 0..99
1 more shapes without text or variables
*)

(* Visualisation SETUP
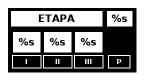
rectangle at (2,2)-(95,19): text "ETAPA"
rectangle at (98,2)-(125,19): text "%s"; shows .IHM_INT_ETAPAS
rectangle at (4,23)-(33,45): text "%s"; shows .IHM_INT_ATIVOS[1]; editable 0..15
rectangle at (35,23)-(64,45): text "%s"; shows .IHM_INT_ATIVOS[2]; editable 0..15
rectangle at (66,23)-(95,45): text "%s"; shows .IHM_INT_ATIVOS[3]; editable 0..15
rectangle at (4,47)-(33,60): text "I"
rectangle at (35,47)-(64,60): text "II"
rectangle at (66,47)-(95,60): text "III"
rectangle at (100,47)-(122,60): text "P"
1 more shapes without text or variables
1 elements of other kinds (tables, trends, ...) not read
*)
